FUNCTION_BLOCK FB_BaseDiverter IMPLEMENTS I_Actuator
VAR
    bEnabled : BOOL;
    bActive : BOOL;
END_VAR

METHOD Disable : bool
VAR_INPUT
END_VAR
bEnabled := FALSE;
bActive := FALSE;
END_METHOD

METHOD Enable : bool
VAR_INPUT
END_VAR
bEnabled := TRUE;
END_METHOD

METHOD Init : bool
VAR_INPUT
END_VAR
END_METHOD

METHOD Start : bool
VAR_INPUT
END_VAR
IF bEnabled THEN
    bActive := TRUE;
END_IF
END_METHOD

METHOD Stop : bool
VAR_INPUT
END_VAR
bActive := FALSE;
END_METHOD

METHOD Update : bool
VAR_INPUT
END_VAR
END_METHOD

END_FUNCTION_BLOCK

(* stored: Version 1.1.0.1
   POU FB_BaseDiverter: Id {6ac4f98e-5856-4f72-bcb6-80ab840b0b86}, SpecialFunc None
   Method Disable: Id {a80962d5-c493-4df1-96b8-45274d7493d3}
   Method Enable: Id {bc6f8fcd-9ef2-4260-aced-3e6b1c7bd973}
   Method Init: Id {94c0a34b-9fae-402c-8f08-cf7bc5df61fb}
   Method Start: Id {b70e79c5-5d4e-4623-b435-ebf672011738}
   Method Stop: Id {f383ec56-0136-435e-9a68-7b6f7ccccdc9}
   Method Update: Id {1182cb1e-ebb7-4c3e-a294-e7831cf0baf2} *)
